{attribute addProperty BoxType "EK1122-0000-0018"}
{attribute addProperty Id "Beckhoff_EPP1xxxsub_EK1100EK1100_179A0949162A_0001_EPP1004_0061_0016EPP1004_5A15FBDA648A_0002_EPP1008_0001_0016EPP1008_C6161DDF9612A_0003_EPP1008_0001_0017EPP1008_C6161DDF9612A_0004_EPP1008_0002_0016EPP1008_C6161DDF9612A_0005_EPP1008_0002_0017EPP1008_C6161DDF9612A_0006_EPP1008_0022_0016EPP1008_C6161DDF9612A_0007_EPP1018_0001_0016EPP1018_C6161DDF9612A_0008_EPP1018_0001_0017EPP1018_C6161DDF9612A_0009_EPP1018_0002_0016EPP1018_C6161DDF9612A_0010_EPP1018_0002_0017EPP1018_C6161DDF9612A_0011_EPP1111_0000_0016EPP1111_BAD6F5C211214A_0012_EPP1111_0000_0017EPP1111_BAD6F5C211214A_0013_EPP1111_0000_0018EPP1111_BAD6F5C211214A_0014_EPP1258_0001_0016EPP1258_402FC40E44856A_0015_EPP1258_0001_0017EPP1258_402FC40E44856A_0016_EPP1258_0002_0016EPP1258_402FC40E44856A_0017_EPP1258_0002_0017EPP1258_402FC40E44856A_0018_EPP1321_0060_0016A_0018_EPP1321_0060_0016_E0E6A0B72816352"}
{attribute addProperty CRC "2786740649"}
{attribute addProperty SizeInBites "5888"}
{attribute addProperty SizeInBytes "736"}
TYPE Beckhoff_EPP1xxxEK1122_A61A49A9 EXTENDS EK1122_179A0949 :
STRUCT
	{attribute addProperty Name "Beckhoff_EPP1xxxsub_EK1100"}
	Beckhoff_EPP1xxxsub_EK1100 : EK1100_179A0949;
	{attribute addProperty Name "A_0001_EPP1004_0061_0016"}
	A_0001_EPP1004_0061_0016 : EPP1004_5A15FBDA;
	{attribute addProperty Name "A_0002_EPP1008_0001_0016"}
	A_0002_EPP1008_0001_0016 : EPP1008_C6161DDF;
	{attribute addProperty Name "A_0003_EPP1008_0001_0017"}
	A_0003_EPP1008_0001_0017 : EPP1008_C6161DDF;
	{attribute addProperty Name "A_0004_EPP1008_0002_0016"}
	A_0004_EPP1008_0002_0016 : EPP1008_C6161DDF;
	{attribute addProperty Name "A_0005_EPP1008_0002_0017"}
	A_0005_EPP1008_0002_0017 : EPP1008_C6161DDF;
	{attribute addProperty Name "A_0006_EPP1008_0022_0016"}
	A_0006_EPP1008_0022_0016 : EPP1008_C6161DDF;
	{attribute addProperty Name "A_0007_EPP1018_0001_0016"}
	A_0007_EPP1018_0001_0016 : EPP1018_C6161DDF;
	{attribute addProperty Name "A_0008_EPP1018_0001_0017"}
	A_0008_EPP1018_0001_0017 : EPP1018_C6161DDF;
	{attribute addProperty Name "A_0009_EPP1018_0002_0016"}
	A_0009_EPP1018_0002_0016 : EPP1018_C6161DDF;
	{attribute addProperty Name "A_0010_EPP1018_0002_0017"}
	A_0010_EPP1018_0002_0017 : EPP1018_C6161DDF;
	{attribute addProperty Name "A_0011_EPP1111_0000_0016"}
	A_0011_EPP1111_0000_0016 : EPP1111_BAD6F5C2;
	{attribute addProperty Name "A_0012_EPP1111_0000_0017"}
	A_0012_EPP1111_0000_0017 : EPP1111_BAD6F5C2;
	{attribute addProperty Name "A_0013_EPP1111_0000_0018"}
	A_0013_EPP1111_0000_0018 : EPP1111_BAD6F5C2;
	{attribute addProperty Name "A_0014_EPP1258_0001_0016"}
	A_0014_EPP1258_0001_0016 : EPP1258_402FC40E;
	{attribute addProperty Name "A_0015_EPP1258_0001_0017"}
	A_0015_EPP1258_0001_0017 : EPP1258_402FC40E;
	{attribute addProperty Name "A_0016_EPP1258_0002_0016"}
	A_0016_EPP1258_0002_0016 : EPP1258_402FC40E;
	{attribute addProperty Name "A_0017_EPP1258_0002_0017"}
	A_0017_EPP1258_0002_0017 : EPP1258_402FC40E;
	{attribute addProperty Name "A_0018_EPP1321_0060_0016"}
	A_0018_EPP1321_0060_0016 : A_0018_EPP1321_0060_0016_E0E6A0B7;
END_STRUCT
END_TYPE

(* stored: Version 1.2.0.0, ProductVersion 3.1.4024.9
   DUT Beckhoff_EPP1xxxEK1122_A61A49A9: Id {0ea4de2d-bd3c-4321-94a0-b153f19c5bef} *)
